// TIA Portal V17 export
// export: Created 2024-09-15T12:30:11.4351515Z, ExportSetting WithDefaults, DisplayName Totally Integrated Automation Portal, DisplayVersion V17, DisplayName TIA Portal Openness, DisplayVersion V17, DisplayName TIA Portal Version Control Interface, DisplayVersion V17, DisplayName STEP 7 Professional, DisplayVersion V17, DisplayName STEP 7 Safety, DisplayVersion V17, DisplayName WinCC Professional, DisplayVersion V17
DATA_BLOCK "MPO_Tracking_DB"   // DB50
VERSION : 0.1
// stored: AutoNumber true, DBAccessibleFromOPCUA true, DBAccessibleFromWebserver true, InstanceOfName MPO_Tracking, InstanceOfType FB
"MPO_Tracking"
   // VAR
   //    Location : String;
   // END_VAR
BEGIN
END_DATA_BLOCK
